{attribute 'qualified_only'}
{attribute 'strict'}
TYPE PisaPulseCommMode :
(
	Offline :=0,
	Unidirectional := 1,
	Bidirectional :=2
	
);
END_TYPE

(* stored: Version 1.1.0.1, ProductVersion 3.1.4024.15
   EnumerationTextList PisaPulseCommMode: Id {7b5bee69-3728-4b92-afd8-8e73f6a3032c} *)
